// TIA Portal V20 export
DATA_BLOCK "CallEquipment_DB"   // DB95
{ DB_Accessible_From_OPC_UA := 'FALSE' }
// stored: AssignedProDiagFB Unit1.Em7.ProDiag, DBAccessibleFromOPCUA false, DBAccessibleFromWebserver false, InstanceOfName Unit1.Em7.CallEquipment, InstanceOfType FB, Namespace Unit1.Em7
"Unit1.Em7.CallEquipment"
   // VAR_INPUT
   //    ZoneOperationEnable { ExternalWritable := 'False'} : "LWONIK_typeSafetyZoneManualOperation";
   //    unitEnableControlInterfaces { ExternalWritable := 'False'} : "LAF_typeEnableControlInterfaces";
   //    commandExcute { ExternalWritable := 'False'} : Bool;
   // END_VAR
   // VAR_IN_OUT
   //    unitStatus : "LAF_typeUnitStatus";
   //    emFeedback : "LUC_typeEmFeedback";
   //    unitAlarmDB : "LAF_typeAlarms";
   // END_VAR
   // VAR
   //    instSequenceConveyor { ExternalWritable := 'False'} : "Unit1.Em7.Sequence_1_Conveyor";
   //    instSequenceNgKicker { ExternalWritable := 'False'} : "Unit1.Em7.Sequence_2_Kicker";
   //    instSequencePassKicker { ExternalWritable := 'False'} : "Unit1.Em7.Sequence_2_Kicker";
   //    instSequenceQrRreader_Stack1 { ExternalWritable := 'False'} : "Unit1.Em7.Sequence_3_QrReader";
   //    instSequenceQrRreader_Stack2 { ExternalWritable := 'False'} : "Unit1.Em7.Sequence_3_QrReader";
   //    instSequenceSTKInterface_Stack1 { ExternalWritable := 'False'} : "Unit1.Em7.Sequence_4_STKInterface";
   //    instSequenceSTKInterface_Stack2 { ExternalWritable := 'False'} : "Unit1.Em7.Sequence_4_STKInterface";
   //    instConveyorInitializedJob1 { ExternalWritable := 'False'} : "LAF_SelectJob";
   //    instConveyorMotionAutoJob2 { ExternalWritable := 'False'} : "LAF_SelectJob";
   //    instConveyorPitchAutoJob3 { ExternalWritable := 'False'} : "LAF_SelectJob";
   //    instConveyorReWorkReqJob8 { ExternalWritable := 'False'} : "LAF_SelectJob";
   //    instConveyorVisionReqJob9 { ExternalWritable := 'False'} : "LAF_SelectJob";
   //    instConveyorGaugeRnRType1Job10 { ExternalWritable := 'False'} : "LAF_SelectJob";
   //    instNgKickerInitializedJob1 { ExternalWritable := 'False'} : "LAF_SelectJob";
   //    instNgKickerAutoJob2 { ExternalWritable := 'False'} : "LAF_SelectJob";
   //    instPassKickerInitializedJob1 { ExternalWritable := 'False'} : "LAF_SelectJob";
   //    instPassKickerAutoJob2 { ExternalWritable := 'False'} : "LAF_SelectJob";
   //    instSTK1QrReadInitializedJob1 { ExternalWritable := 'False'} : "LAF_SelectJob";
   //    instSTK1QrReadAutoJob2 { ExternalWritable := 'False'} : "LAF_SelectJob";
   //    instSTK2QrReadInitializedJob1 { ExternalWritable := 'False'} : "LAF_SelectJob";
   //    instSTK2QrReadAutoJob2 { ExternalWritable := 'False'} : "LAF_SelectJob";
   //    instSTK1InterfaceInitializedJob1 { ExternalWritable := 'False'} : "LAF_SelectJob";
   //    instSTK1InterfaceAutoJob2 { ExternalWritable := 'False'} : "LAF_SelectJob";
   //    instSTK2InterfaceInitializedJob1 { ExternalWritable := 'False'} : "LAF_SelectJob";
   //    instSTK2InterfaceAutoJob2 { ExternalWritable := 'False'} : "LAF_SelectJob";
   //    instCmNgKickerAxisZ { ExternalWritable := 'False'} : "LBC_AxisControl_TecPlcCn";
   //    instCmPassKickerAxisZ { ExternalWritable := 'False'} : "LBC_AxisControl_TecPlcCn";
   //    instCmCutConveyorAxisB { ExternalWritable := 'False'} : "LBC_AxisControl_TecPlcCn";
   //    instCmNgConveyorAxisB { ExternalWritable := 'False'} : "LBC_AxisControl_TecPlcCn";
   //    instCmStack1ConveyorAxisB { ExternalWritable := 'False'} : "LBC_AxisControl_TecPlcCn";
   //    instCmStack2ConveyorAxisB { ExternalWritable := 'False'} : "LBC_AxisControl_TecPlcCn";
   //    instCmConveyorVirtualAxisB { ExternalWritable := 'False'} : "LBC_AxisControl_TecPlcCn";
   //    instCmCutConveyorRingBlow { ExternalWritable := 'False'} : "LBC_SinaSpeedCn";
   //    instCmNgConveyorRingBlow { ExternalWritable := 'False'} : "LBC_SinaSpeedCn";
   //    instCmStack2ConveyorRingBlow { ExternalWritable := 'False'} : "LBC_SinaSpeedCn";
   //    instcmNgBoxLockCylinderUpDown { ExternalWritable := 'False'} : "LBC_TwoWayActuatorCn";
   //    instCmNgBoxDetectSensor { ExternalWritable := 'False'} : "LBC_DigitalSignalCn";
   //    instCmNgBoxFullSensor { ExternalWritable := 'False'} : "LBC_DigitalSignalCn";
   //    instCmNgKickerDetectSensor { ExternalWritable := 'False'} : "LBC_DigitalSignalCn";
   //    instCmPassKickerDetectSensor { ExternalWritable := 'False'} : "LBC_DigitalSignalCn";
   //    instCmStack1ConveyorElectrodeDetectSensor { ExternalWritable := 'False'} : "LBC_DigitalSignalCn";
   //    instCmStack2ConveyorElectrodeDetectSensor { ExternalWritable := 'False'} : "LBC_DigitalSignalCn";
   //    instCmStack1QRreader { ExternalWritable := 'False'} : "LER_QRread_SRX300";
   //    instCmStack2QRreader { ExternalWritable := 'False'} : "LER_QRread_SRX300";
   //    instCmNgKickerAxisControlInterlockSummary { ExternalWritable := 'False'} : "LER_AxisControl_InterlockSummary";
   //    instCmPassKickerAxisControlInterlockSummary { ExternalWritable := 'False'} : "LER_AxisControl_InterlockSummary";
   //    instCmCutConveyorAxisControlInterlockSummary { ExternalWritable := 'False'} : "LER_AxisControl_InterlockSummary";
   //    instCmNgConveyorAxisControlInterlockSummary { ExternalWritable := 'False'} : "LER_AxisControl_InterlockSummary";
   //    instCmStack1ConveyorAxisControlInterlockSummary { ExternalWritable := 'False'} : "LER_AxisControl_InterlockSummary";
   //    instCmStack2ConveyorAxisControlInterlockSummary { ExternalWritable := 'False'} : "LER_AxisControl_InterlockSummary";
   //    instCmConveyorVirtualAxisControlInterlockSummary { ExternalWritable := 'False'} : "LER_AxisControl_InterlockSummary";
   //    instServoTorqueCal_DR10 { ExternalWritable := 'False'} : "LER_ServoTorqueCal";
   //    instServoTorqueCal_DR11 { ExternalWritable := 'False'} : "LER_ServoTorqueCal";
   //    instServoTorqueCal_DR12 { ExternalWritable := 'False'} : "LER_ServoTorqueCal";
   //    instServoTorqueCal_DR13 { ExternalWritable := 'False'} : "LER_ServoTorqueCal";
   //    instServoTorqueCal_DR14 { ExternalWritable := 'False'} : "LER_ServoTorqueCal";
   //    instServoTorqueCal_DR15 { ExternalWritable := 'False'} : "LER_ServoTorqueCal";
   //    instLDrv701ControlNgKickerAxisZ { ExternalWritable := 'False'} : "LDrvSafe_SinaTlg701Control";
   //    instLDrv701StatusNgKickerAxisZ { ExternalWritable := 'False'} : "LDrvSafe_SinaTlg701Status";
   //    instLDrv701ControlPassKickerAxisZ { ExternalWritable := 'False'} : "LDrvSafe_SinaTlg701Control";
   //    instLDrv701StatusPassKickerAxisZ { ExternalWritable := 'False'} : "LDrvSafe_SinaTlg701Status";
   //    statUnitStatus { ExternalWritable := 'False'} : "LAF_typeUnitStatus";
   //    statAllBrakeTest { ExternalWritable := 'False'} : "LER_typeBrakeTestUnitCommands";
   //    instManageAlarms { ExternalWritable := 'False'} : "LAF_ManageAlarms";
   //    instEventsPFE { ExternalWritable := 'False'} : "Unit1.Em7.EventsPFE";
   //    statPulse { ExternalWritable := 'False'} : Array[0..99] of Bool;
   //    statTonTimer { ExternalWritable := 'False'} : Array[0..99] of TON_TIME;
   //    statTofTimer { ExternalWritable := 'False'} : Array[0..99] of TOF_TIME;
   //    statEnableManualCmds { ExternalWritable := 'False'} : Bool;
   //    statJobSummary { ExternalWritable := 'False'} : "LAF_typeJobStatus";
   //    statRunOutCheck { ExternalWritable := 'False'} : Struct
   //       CutConveyor : Bool;
   //       NgConveyor : Bool;
   //       Stack1Conveyor : Bool;
   //       Stack2Conveyor : Bool;
   //       RunOutComplete : Bool;
   //    END_STRUCT;
   //    statSafeStateCheck { ExternalWritable := 'False'} : Struct
   //       Conveyor : Bool;
   //       NgKicker : Bool;
   //       PassKicker : Bool;
   //       Stack1QrReader : Bool;
   //       Stkac2QrReader : Bool;
   //       Stack1Interrface : Bool;
   //       Stack2Interface : Bool;
   //    END_STRUCT;
   //    statPitchDistance { ExternalWritable := 'False'} : LReal;
   //    instCVFullChargeCheckCMD { ExternalWritable := 'False'} : "LAF_SelectJob";
   //    instStackGaugeRnRJob12 { ExternalWritable := 'False'} : "LAF_SelectJob";
   //    DataClearCheck { ExternalWritable := 'False'} : Bool;
   //    RunOutCMD { ExternalWritable := 'False'} : Bool;
   //    StackRunOutCMD { ExternalWritable := 'False'} : Bool;
   //    ParameterChangeMonitor_Instance { ExternalWritable := 'False'} : "Unit1.Em7.ParameterChangeMonitor";
   //    ParaChangeRunOut { ExternalWritable := 'False'} : Bool;
   //    ParameterChanged { ExternalWritable := 'False'} : Bool;
   //    statCutSavePosition { ExternalWritable := 'False'} : LReal;
   //    statNGSavePosition { ExternalWritable := 'False'} : LReal;
   //    statStack1SavePosition { ExternalWritable := 'False'} : LReal;
   //    statStack2SavePosition { ExternalWritable := 'False'} : LReal;
   //    statCutSub { ExternalWritable := 'False'} : LReal;
   //    statNGSub { ExternalWritable := 'False'} : LReal;
   //    statStack1Sub { ExternalWritable := 'False'} : LReal;
   //    statStack2Sub { ExternalWritable := 'False'} : LReal;
   //    statCutSub_1 { ExternalWritable := 'False'} : LReal;
   //    statNGSub_1 { ExternalWritable := 'False'} : LReal;
   //    statStack1Sub_1 { ExternalWritable := 'False'} : LReal;
   //    statStack2Sub_1 { ExternalWritable := 'False'} : LReal;
   //    PitchSubComp { ExternalWritable := 'False'} : Bool;
   //    PitchCutNG { ExternalWritable := 'False'} : Bool;
   //    PitchNgNG { ExternalWritable := 'False'} : Bool;
   //    PitchStack1NG { ExternalWritable := 'False'} : Bool;
   //    PitchStack2NG { ExternalWritable := 'False'} : Bool;
   //    PitchCutOK { ExternalWritable := 'False'} : Bool;
   //    PitchNgOK { ExternalWritable := 'False'} : Bool;
   //    PitchStack1OK { ExternalWritable := 'False'} : Bool;
   //    PitchStack2OK { ExternalWritable := 'False'} : Bool;
   //    PitchUpdate { ExternalWritable := 'False'} : Bool;
   //    RecoveryStep { ExternalWritable := 'False'} : Int;
   //    citi_Ptrig : Array[0..20] of Bool;
   //    citiTon : Array[0..20] of TON_TIME;
   //    citi : Time;
   //    citiTest : Array[0..20] of Bool;
   // END_VAR
BEGIN
END_DATA_BLOCK
